FUNCTION_BLOCK AdsSocket
VAR_STAT
	localPrgName : STRING; //:= GVL.localPrgName;
	localNetId : T_AmsNetId; //:= GVL.localAmsNetId;
	localPort : T_AmsPort; //:= GVL.localAmsPort;
END_VAR
VAR
	remotePrgName : STRING;
	remoteNetId : T_AmsNetId;
	remotePort : T_AmsPort;
END_VAR
VAR
	adsReadSymbol : FB_ReadAdsSymByName;
	adsWriteSymbol : FB_WriteAdsSymByName;
END_VAR

METHOD close : BOOL
remotePrgName := '';
remoteNetId := '';
remotePort := 0;
END_METHOD

METHOD open : BOOL
VAR_INPUT
	newLocalPrgName : STRING;
	newLocalNetId : T_AmsNetId;
	newLocalPort : T_AmsPort;
END_VAR
localPrgName := newLocalPrgName;
localNetId := newLocalNetId;
localPort := newLocalPort;

adsWriteSymbol.sNetId:= remoteNetId;
adsWriteSymbol.nPort:= remotePort;
END_METHOD

METHOD read : BOOL
VAR_INPUT
	symbol : STRING;
	buffer : PVOID;
	symbolSize : UDINT;
END_VAR
adsReadSymbol(
	bRead:= , 
	sNetId:= remoteNetId, 
	nPort:= remotePort, 
	sVarName:= symbol, 
	nDestAddr:= buffer, 
	nLen:= symbolSize, 
	tTimeout:= , 
	eComMode:= , 
	bClearOnError:= TRUE, 
	bBusy=> , 
	bError=> , 
	nErrorId=> );
	
adsReadSymbol.bRead := FALSE;
END_METHOD

METHOD ready : BOOL
ready := (
	remotePrgName <> '' AND
	remoteNetId <> '' AND
	remotePort <> 0);
END_METHOD

METHOD setup : BOOL
localPrgName := '';
localNetId := '';
localPort := 0;

//fill these values with data
END_METHOD

METHOD write : BOOL
VAR_INPUT
	symbol : STRING;
	data : PVOID;
	dataSize : UDINT;
END_VAR
adsWriteSymbol(
	bWrite:= TRUE, 
	sNetId:= remoteNetId, 
	nPort:= remotePort, 
	sVarName:= symbol, 
	nSrcAddr:= data, 
	nLen:= dataSize, 
	tTimeout:= , 
	eComMode:= , 
	bBusy=> , 
	bError=> , 
	nErrorId=> );
	
adsWriteSymbol.bWrite := FALSE;
END_METHOD

END_FUNCTION_BLOCK

(* stored: Version 1.1.0.1, ProductVersion 3.1.4024.11
   POU AdsSocket: Id {94b06c8f-6363-4f38-8057-d0f2ec092ac9}, SpecialFunc None
   Method close: Id {5b9b3a4a-f4db-4662-8e31-880b17578695}
   Method open: Id {41dcc539-006b-4672-ab53-559a081cb5fc}
   Method read: Id {76310918-f166-49dc-9eaa-fa797266bfbf}
   Method ready: Id {6481e89a-6c18-4ef9-9fbf-31fc0017edf1}
   Method setup: Id {a4b0e4a8-298b-4495-939e-427add857afc}
   Method write: Id {78b7348b-168f-4aaf-82b1-6907845ef997} *)
